// TIA Portal V20 export
TYPE "LER_typeUnitData"
// stored: Access Published
   STRUCT
      QrReadID : String[64];
      VisionAlign : "LER_typeVisionAlignData";
      VisionGap : "LER_typeVisionGapData";
   END_STRUCT;
END_TYPE
